// TIA Portal V20 export
DATA_BLOCK "instRfidAntenaLeft"   // DB67
// stored: AssignedProDiagFB ProDiag, InstanceOfName LER_RFID, InstanceOfType FB
"LER_RFID"
   // VAR_INPUT
   //    enable : Bool;
   //    enableManualCmds : Bool;
   //    bobinChuck : Bool;
   // END_VAR
   // VAR_OUTPUT
   //    error : Bool;
   //    status : DWord;
   // END_VAR
   // VAR_IN_OUT
   //    RFID_Chanel : TO_IDENT;
   //    IdentRfAntena : "LSicar_typeIdentInterfaceHmi";
   //    moduleInterface : "LER_typeRFIDInterface";
   // END_VAR
   // VAR
   //    instResetReader : Reset_Reader;
   //    instRead : Read;
   //    instWrite : Write;
   //    instInventory : Inventory;
   //    statResetReaderUDT : "LER_typeResetReaderUDT";
   //    statReadUDT : "LER_typeReadWriteUDT";
   //    statWriteUDT : "LER_typeReadWriteUDT";
   //    statInventoryUDT : "LER_typeInventoryUDT";
   //    statResultRFIDReset : Bool;
   //    statPulse : Array[0..9] of Bool;
   //    statTonTimer : TON_TIME;
   //    statBobinData : IID_IN_I_81;
   //    statRFID_str : String[32];
   //    statEPCID_str : String[32];
   //    statHi : Byte;
   //    statLo : Byte;
   //    statHexArray : Array[0..15] of Char;
   // END_VAR
BEGIN
END_DATA_BLOCK
